PROGRAM prgComEffIO
VAR
	fbCom		: FB_MqttCommunicator;
END_VAR

fbCom(
	bConnect:= TRUE, 
	sUserName:= 'd7aecbab-7f4e-4acb-b33b-24861f013074', 
	sUserPassword:= '3abb15af-0787-45ea-b3af-d708d75008a0', 
	eSavePositionCertificate:= eSavePositionOnPLC.ePostionHardDisk, 
	bConnected=> , 
	bError=> , 
	hrErrorCode=> , 
	eConnectionState=> , 
	eErrorMessage_Out=> );

END_PROGRAM

(* stored: Version 1.1.0.1, ProductVersion 3.1.4024.11
   POU prgComEffIO: Id {cbcd318b-bf51-484c-bcaa-d6efcdf43fe3}, SpecialFunc None *)
